ABB RobotStudio station: RobMan1.rsstn

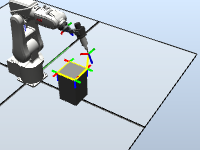
Station RobMan1 (saved by RobotStudio 6.6.7701.1025)
Controller Sistema1
  mechanical unit ROB_1: IRB120_3_58__01, 6 joints, base frame (0, 0, 0) mm
Layout (positions relative to the parent item):
  - IRB120_3_58__01 [mechanism, from Robots\IRB120_3_58_G_01.rslib] at (0, 0, 0) mm; joint values [0, 0, 0, 0, 0.5236, 0] (rad or m)
  - MyTool [mechanism, from Training Objects\myTool.rslib] at (364.35, 0, 594) mm, rotated rx 180 ry 60 rz 180 deg
  - Pieza_2 [part]
Attachment: MyTool is attached to IRB120_3_58__01 / Link6
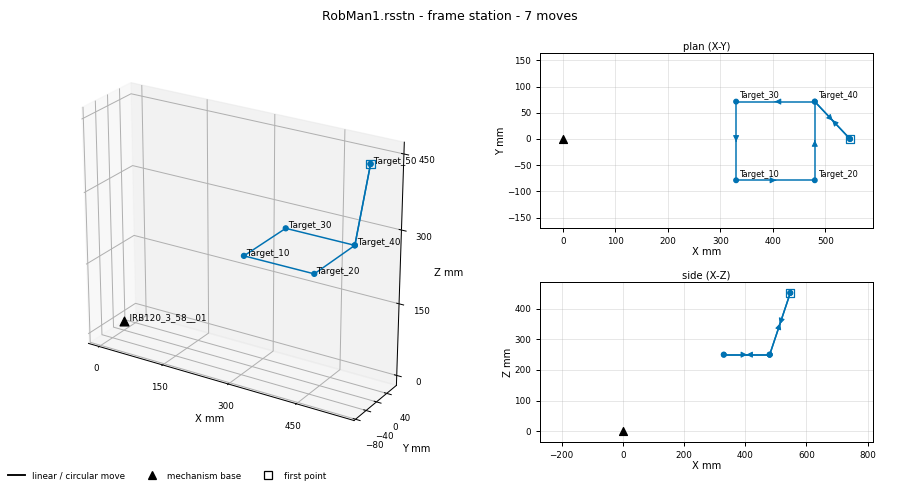
[picture p0: tool path of RobMan1.rsstn in frame station, 7 of 7 moves have a stored position in this frame; points joined in program order, loops and branches not executed]
Targets, tools, work objects and paths stored in the station, written as RAPID:
! task T_ROB1
MODULE CalibData
  PERS tooldata MyTool:=[TRUE,[[31.792631019,0,229.638935148],[0.945518576,0,0.325568154,0]],[1,[0,0,1],[1,0,0,0],0,0,0]];
ENDMODULE

! task T_ROB1
MODULE Module1
  CONST robtarget Target_10:=[[330.118,-78.723,250],[0,-0.707106781,0.707106781,0],[-1,0,-2,0],[9E+09,9E+09,9E+09,9E+09,9E+09,9E+09]];
  CONST robtarget Target_20:=[[480.118,-78.723,250],[0,0.707106781,0.707106781,0],[0,-1,1,0],[9E+09,9E+09,9E+09,9E+09,9E+09,9E+09]];
  CONST robtarget Target_30:=[[330.118,71.277,250],[0,0,1,0],[0,-1,0,0],[9E+09,9E+09,9E+09,9E+09,9E+09,9E+09]];
  CONST robtarget Target_40:=[[480.118,71.277,250],[0,0.707106781,0.707106781,0],[0,-1,1,0],[9E+09,9E+09,9E+09,9E+09,9E+09,9E+09]];
  CONST robtarget Target_50:=[[547.330665099,0,451.64730631],[0.190808996,0,0.981627183,0],[-1,0,-1,0],[9E+09,9E+09,9E+09,9E+09,9E+09,9E+09]];
  PROC Path_10()
    MoveL Target_50,v1000,fine,MyTool\WObj:=wobj0;
    MoveL Target_40,v500,fine,MyTool\WObj:=wobj0;
    MoveL Target_30,v500,fine,MyTool\WObj:=wobj0;
    MoveL Target_10,v500,fine,MyTool\WObj:=wobj0;
    MoveL Target_20,v500,z0,MyTool\WObj:=wobj0;
    MoveL Target_40,v500,fine,MyTool\WObj:=wobj0;
    MoveL Target_50,v1000,fine,MyTool\WObj:=wobj0;
  ENDPROC
ENDMODULE

